(* IEC 61131-3 sources: ArfBotOS/Codesys-4/ArfBotOS.fbsdev/Application.iecapp^/FUN/template/FB_PackML.fb.st^/transition, 10 files *)

(* ---- M_Aborting.meth.st ---- *)
METHOD PROTECTED M_Aborting : BOOL
VAR_INPUT
END_VAR

_StateTimer.IN:=TRUE;

IF _StateTimer.Q THEN
	_StateTimer.IN:=FALSE;
	M_StateComplete();
END_IF
END_METHOD

(* ---- M_Clearing.meth.st ---- *)
METHOD PROTECTED M_Clearing : BOOL
VAR_INPUT
END_VAR

_StateTimer.IN:=TRUE;

IF _StateTimer.Q THEN
	_StateTimer.IN:=FALSE;
	M_StateComplete();
END_IF
END_METHOD

(* ---- M_Completing.meth.st ---- *)
METHOD PROTECTED M_Completing : BOOL
VAR_INPUT
END_VAR

_StateTimer.IN:=TRUE;

IF _StateTimer.Q THEN
	_StateTimer.IN:=FALSE;
	M_StateComplete();
END_IF
END_METHOD

(* ---- M_Holding.meth.st ---- *)
METHOD PROTECTED M_Holding : BOOL
VAR_INPUT
END_VAR

_StateTimer.IN:=TRUE;

IF _StateTimer.Q THEN
	_StateTimer.IN:=FALSE;
	M_StateComplete();
END_IF
END_METHOD

(* ---- M_Resetting.meth.st ---- *)
METHOD PROTECTED M_Resetting : BOOL
VAR_INPUT
END_VAR

_StateTimer.IN:=TRUE;

IF _StateTimer.Q THEN
	_StateTimer.IN:=FALSE;
	M_StateComplete();
END_IF
END_METHOD

(* ---- M_Starting.meth.st ---- *)
METHOD PROTECTED M_Starting : BOOL
VAR_INPUT
END_VAR

_StateTimer.IN:=TRUE;

IF _StateTimer.Q THEN
	_StateTimer.IN:=FALSE;
	M_StateComplete();
END_IF
END_METHOD

(* ---- M_Stopping.meth.st ---- *)
METHOD PROTECTED M_Stopping : BOOL
VAR_INPUT
END_VAR

_StateTimer.IN:=TRUE;

IF _StateTimer.Q THEN
	_StateTimer.IN:=FALSE;
	M_StateComplete();
END_IF
END_METHOD

(* ---- M_Suspending.meth.st ---- *)
METHOD PROTECTED M_Suspending : BOOL
VAR_INPUT
END_VAR

_StateTimer.IN:=TRUE;

IF _StateTimer.Q THEN
	_StateTimer.IN:=FALSE;
	M_StateComplete();
END_IF
END_METHOD

(* ---- M_Unholding.meth.st ---- *)
METHOD PROTECTED M_Unholding : BOOL
VAR_INPUT
END_VAR

_StateTimer.IN:=TRUE;

IF _StateTimer.Q THEN
	_StateTimer.IN:=FALSE;
	M_StateComplete();
END_IF
END_METHOD

(* ---- M_UnSuspending.meth.st ---- *)
METHOD PROTECTED M_UnSuspending : BOOL
VAR_INPUT
END_VAR

_StateTimer.IN:=TRUE;

IF _StateTimer.Q THEN
	_StateTimer.IN:=FALSE;
	M_StateComplete();
END_IF
END_METHOD
